// TIA Portal project "BibiteFB" (V16)

(* hardware
DEVICE "S7-1200 station_1"  S7-1200 Station
   slot 0: "Telaio di montaggio_0"  S7-1200 Rack  Rack  V1.0
   slot 1: "PLC_1"  CPU 1214C DC/DC/DC  6ES7 214-1AG40-0XB0  V4.4
*)

// ===== PLC "PLC_1"  CPU 1214C DC/DC/DC =====

VAR_GLOBAL   // PLC tag table "Tabella delle variabili standard"
   "Moneta" AT %I0.0 : Bool;
   "FineCorsaA" AT %I0.1 : Bool;
   "FineCorsaB" AT %I0.2 : Bool;
   "BibitaPresente" AT %I0.3 : Bool;
   "Prelievo" AT %M0.0 : Bool;
   "SA" AT %Q0.1 : Bool;
   "SB" AT %Q0.2 : Bool;
   "BLOCCA" AT %Q0.3 : Bool;
END_VAR

VAR_GLOBAL CONSTANT   // PLC tag table "Tabella delle variabili standard"
   "Delay" : Time := T#5s;
END_VAR

DATA_BLOCK "DistributoreBibite_DB"   // DB1
{ S7_Optimized_Access := 'TRUE' }
VERSION : 0.1
// stored: InstanceOfName DistributoreBibite
"DistributoreBibite"
BEGIN
END_DATA_BLOCK

FUNCTION_BLOCK "DistributoreBibite"   // FB1, LAD
{ S7_Optimized_Access := 'TRUE' }
VERSION : 0.1
   VAR_INPUT
      Moneta : Bool;
      FineCorsaA : Bool;
      FineCorsaB : Bool;
      BibitaPresente : Bool;
      Delay : Time := T#5s;
   END_VAR
   VAR_OUTPUT
      SA : Bool;
      SB : Bool;
      BLOCCA : Bool;
   END_VAR
   VAR_IN_OUT
      Prelievo : Bool;
   END_VAR
   VAR RETAIN
      HOME : Bool := true;
      ConsegnaBibita : Bool;
      RientroSB : Bool;
      NuovaBibita : Bool;
      RientroSA : Bool;
      Attesa : Bool;
   END_VAR
   VAR
      IEC_Timer_0_Instance : TON_TIME;
      IEC_Timer_0_Instance_1 : TON_TIME;
   END_VAR
BEGIN

REGION Network 1
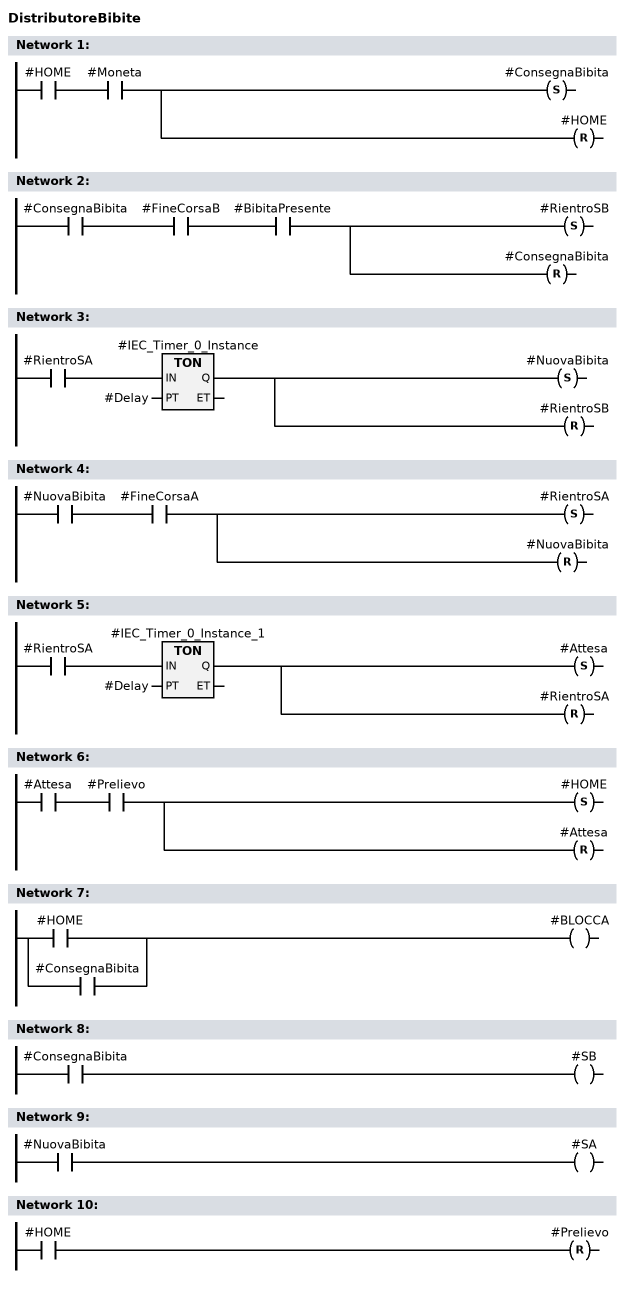
   RUNG wire#powerrail
      Contact( #HOME )
      Contact( #Moneta )
      wire#w1
      S_Coil( #ConsegnaBibita )
   END_RUNG
   RUNG wire#w1
      R_Coil( #HOME )
   END_RUNG
   // the same network as SCL:
   IF #HOME AND #Moneta THEN
       #ConsegnaBibita := TRUE;
       #HOME := FALSE;
   END_IF;
END_REGION

REGION Network 2
   RUNG wire#powerrail
      Contact( #ConsegnaBibita )
      Contact( #FineCorsaB )
      Contact( #BibitaPresente )
      wire#w1
      S_Coil( #RientroSB )
   END_RUNG
   RUNG wire#w1
      R_Coil( #ConsegnaBibita )
   END_RUNG
   // the same network as SCL:
   IF #ConsegnaBibita AND #FineCorsaB AND #BibitaPresente THEN
       #RientroSB := TRUE;
       #ConsegnaBibita := FALSE;
   END_IF;
END_REGION

REGION Network 3
   #IEC_Timer_0_Instance(IN := #RientroSA, PT := #Delay);   // TON
   IF #IEC_Timer_0_Instance.Q THEN
       #NuovaBibita := TRUE;
       #RientroSB := FALSE;
   END_IF;
END_REGION

REGION Network 4
   RUNG wire#powerrail
      Contact( #NuovaBibita )
      Contact( #FineCorsaA )
      wire#w1
      S_Coil( #RientroSA )
   END_RUNG
   RUNG wire#w1
      R_Coil( #NuovaBibita )
   END_RUNG
   // the same network as SCL:
   IF #NuovaBibita AND #FineCorsaA THEN
       #RientroSA := TRUE;
       #NuovaBibita := FALSE;
   END_IF;
END_REGION

REGION Network 5
   #IEC_Timer_0_Instance_1(IN := #RientroSA, PT := #Delay);   // TON
   IF #IEC_Timer_0_Instance_1.Q THEN
       #Attesa := TRUE;
       #RientroSA := FALSE;
   END_IF;
END_REGION

REGION Network 6
   RUNG wire#powerrail
      Contact( #Attesa )
      Contact( #Prelievo )
      wire#w1
      S_Coil( #HOME )
   END_RUNG
   RUNG wire#w1
      R_Coil( #Attesa )
   END_RUNG
   // the same network as SCL:
   IF #Attesa AND #Prelievo THEN
       #HOME := TRUE;
       #Attesa := FALSE;
   END_IF;
END_REGION

REGION Network 7
   RUNG wire#powerrail
      Contact( #HOME )
      wire#w1
      Coil( #BLOCCA )
   END_RUNG
   RUNG wire#powerrail
      Contact( #ConsegnaBibita )
   END_RUNG wire#w1
   // the same network as SCL:
   #BLOCCA := #HOME OR #ConsegnaBibita;
END_REGION

REGION Network 8
   RUNG wire#powerrail
      Contact( #ConsegnaBibita )
      Coil( #SB )
   END_RUNG
   // the same network as SCL:
   #SB := #ConsegnaBibita;
END_REGION

REGION Network 9
   RUNG wire#powerrail
      Contact( #NuovaBibita )
      Coil( #SA )
   END_RUNG
   // the same network as SCL:
   #SA := #NuovaBibita;
END_REGION

REGION Network 10
   RUNG wire#powerrail
      Contact( #HOME )
      R_Coil( #Prelievo )
   END_RUNG
   // the same network as SCL:
   IF #HOME THEN #Prelievo := FALSE; END_IF;
END_REGION
END_FUNCTION_BLOCK

ORGANIZATION_BLOCK "Main"   // OB1, LAD, ProgramCycle
TITLE = "Main Program Sweep (Cycle)"
{ S7_Optimized_Access := 'TRUE' }
VERSION : 0.1
   VAR_INPUT
      Initial_Call : Bool;   // Initial call of this OB
      Remanence : Bool;   // =True, if remanent data are available
   END_VAR
BEGIN

REGION Network 1
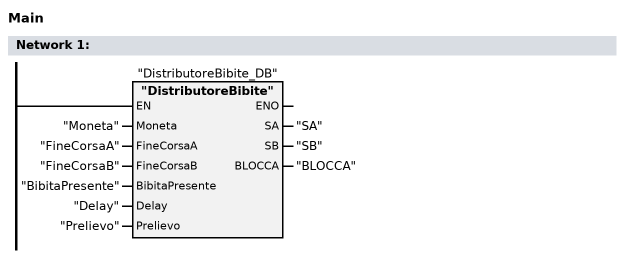
   RUNG wire#powerrail
      "DistributoreBibite_DB"(Moneta := "Moneta", FineCorsaA := "FineCorsaA", FineCorsaB := "FineCorsaB", BibitaPresente := "BibitaPresente", Delay := "Delay", Prelievo := "Prelievo", SA => "SA", SB => "SB", BLOCCA => "BLOCCA")
   END_RUNG
   // the same network as SCL:
   "DistributoreBibite_DB"(Moneta := "Moneta",   // "DistributoreBibite"
                           FineCorsaA := "FineCorsaA",
                           FineCorsaB := "FineCorsaB",
                           BibitaPresente := "BibitaPresente",
                           Delay := "Delay",
                           Prelievo := "Prelievo",
                           SA => "SA",
                           SB => "SB",
                           BLOCCA => "BLOCCA");
END_REGION
END_ORGANIZATION_BLOCK

ORGANIZATION_BLOCK "Hardware interrupt"   // OB40, LAD, HWProcessInterrupt
{ S7_Optimized_Access := 'TRUE' }
VERSION : 0.1
   VAR_INPUT
      LADDR : Hw_Io;   // Hardware identifier
      USI : Word;   // User structure identifier
      IChannel : USInt;   // Interrupt channel number
      EventType : Byte;   // EventType
   END_VAR
BEGIN

REGION Network 1
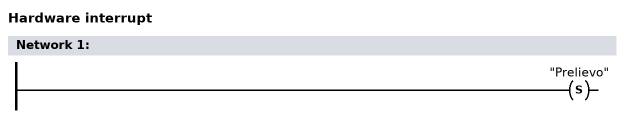
   RUNG wire#powerrail
      S_Coil( "Prelievo" )
   END_RUNG
   // the same network as SCL:
   "Prelievo" := TRUE;
END_REGION
END_ORGANIZATION_BLOCK